FUNCTION_BLOCK EL6751
VAR
	{attribute addProperty Name "Info data"}
	_infoData : InfoDataAdsAoEDC;
END_VAR

END_FUNCTION_BLOCK

(* stored: Version 1.1.0.1, ProductVersion 3.1.4024.9
   POU EL6751: Id {e4751396-d8c5-08a4-0111-a8e2fcf59495}, SpecialFunc None *)
